TYPE ST_RackFeederIO :
STRUCT	
	ioAxisTraverse					: ST_AxisIO;
	ioAxisLift						: ST_AxisIO;
	ioAxisTelescope					: ST_AxisIO;	
	
	ioCarrierPresent				: ST_DigitalInputIO;
	
END_STRUCT
END_TYPE

(* stored: Version 1.1.0.1
   DUT ST_RackFeederIO: Id {2dc2be65-62a3-4716-8617-850d6d1a27f4} *)
